// TIA Portal project "Semaforo V2" (V17)

(* hardware
DEVICE "S7-400 station_1"  S7-400 station
   slot 0: "UR1_0"  UR1  6ES7 400-1TA01-0AA0
   slot 1: "PS 407 4A_1"  PS 407 4A  6ES7 407-0DA02-0AA0
   slot 2: "PLC_1"  CPU 416-3 PN/DP  6ES7 416-3ES07-0AB0  V7.0
      slot 2: "MPI/DP interface_1"  X1
      slot 5: "PROFINET interface_1"  PN-IO
         slot 1: "Port_1"  Port
         slot 2: "Port_2"  Port
*)

// ===== PLC "PLC_1"  CPU 416-3 PN/DP =====

VAR_GLOBAL   // PLC tag table "Default tag table"
   "Tag_1" AT %I0.0 : Bool;
   "Tag_2" AT %Q0.0 : Bool;
   "Tag_3" AT %Q0.1 : Bool;
   "Tag_4" AT %Q0.2 : Bool;
   "Tag_5" AT %Q0.6 : Bool;
   "Tag_6" AT %Q0.5 : Bool;
   "Tag_7" AT %Q0.4 : Bool;
   "Tag_8" AT %Q0.3 : Bool;
   "Tag_9" AT %Q0.7 : Bool;
   "Tag_10" AT %M0.0 : Bool;
   "Tag_11" AT %M0.1 : Bool;
   "Tag_12" AT %I0.1 : Bool;
   "Tag_13" AT %M0.2 : Bool;
   "Tag_14" AT %M0.4 : Bool;
   "Pisca" AT %M1.5 : Bool;
END_VAR

DATA_BLOCK "Block_STL_DB"   // DB1
{ S7_Optimized_Access := 'FALSE' }
VERSION : 0.1
// stored: InstanceOfName Block_STL
"Block_STL"
BEGIN
END_DATA_BLOCK

FUNCTION_BLOCK "Block_STL"   // FB1, STL
{ S7_Optimized_Access := 'FALSE' }
VERSION : 0.1
   VAR_INPUT
      Liga_Desliga : Bool;
      Botao_Pedestre : Bool;
   END_VAR
   VAR_OUTPUT
      A_Vermelho : Bool;
      A_Amarelo : Bool;
      A_Verde : Bool;
      B_Vermelho : Bool;
      B_Amarelo : Bool;
      B_Verde : Bool;
      P_Vermelho : Bool;
      P_Verde : Bool;
   END_VAR
   VAR_TEMP
      Jump : Bool;
      Pedestre1 : Bool;
   END_VAR
BEGIN

REGION Network 1: Semaforos Veículos
         A     #Liga_Desliga;
         AN    "TON5".Q;
         =     "TON2".IN;

         S     #A_Verde;
         S     #B_Vermelho;
         S     #P_Vermelho;

         CALL  TON , "TON2"
         ( IN := ,
           PT := T#20S,
           Q  := ,
           ET :=
         );

         A     "TON2".Q;
         R     #A_Verde;
         S     #A_Amarelo;

         CALL  TON, "TON3"
         ( IN := "TON2".Q,
           PT := T#3S,
           Q  := ,
           ET :=
         );

         A     "TON3".Q;
         R     #A_Amarelo;
         R     #B_Vermelho;
         S     #A_Vermelho;
         S     #B_Verde;

         CALL  TON, "TON4"
         ( IN := "TON3".Q,
           PT := T#20S,
           Q  := ,
           ET :=
         );

         A     "TON4".Q;
         R     #B_Verde;
         S     #B_Amarelo;

         CALL  TON, "TON5"
         ( IN := "TON4".Q,
           PT := T#3S,
           Q  := ,
           ET :=
         );

   //Loop
         AN    #Botao_Pedestre;
         A     "TON5".Q;
         R     #B_Amarelo;
         R     #A_Vermelho;

   //Verificação Pedestre
         A     #Botao_Pedestre;
         A     "TON5".Q;
         =     #Jump;

         A     #Jump;
         JU    pedestre;



   pedestre:S     #Pedestre1;

         A     #Pedestre1;

         S     #A_Vermelho;
         R     #A_Verde;
         R     #A_Amarelo;
         S     #B_Vermelho;
         R     #B_Verde;
         R     #B_Amarelo;
         R     #P_Vermelho;
         S     #P_Verde;


         CALL  TON , "TON6"
         ( IN := #Pedestre1,
           PT := T#20S,
           Q  := ,
           ET :=
         );

         A     "TON6".Q;
         A     "Pisca";
         S     #P_Vermelho;

         A     "TON6".Q;
         AN    "Pisca";
         R     #P_Vermelho;


         A     "TON7".Q;
         S     #P_Vermelho;
         R     #A_Vermelho;
   //   S     #A_Verde
         R     #A_Amarelo;
   //S     #B_Vermelho
         R     #B_Verde;
         R     #B_Amarelo;
         R     #P_Verde;
END_REGION
END_FUNCTION_BLOCK

ORGANIZATION_BLOCK "Main"   // OB1, LAD
TITLE = "Main Program Sweep (Cycle)"
{ S7_Optimized_Access := 'FALSE' }
VERSION : 0.1
   VAR_TEMP
      OB1_EV_CLASS : Byte;   // Bits 0-3 = 1 (Coming event), Bits 4-7 = 1 (Event class 1)
      OB1_SCAN_1 : Byte;   // 1 (Cold restart scan 1 of OB 1), 3 (Scan 2-n of OB 1)
      OB1_PRIORITY : Byte;   // Priority of OB Execution
      OB1_OB_NUMBR : Byte;   // 1 (Organization block 1, OB1)
      OB1_RESERVED_1 : Byte;   // Reserved for system
      OB1_RESERVED_2 : Byte;   // Reserved for system
      OB1_PREV_CYCLE : Int;   // Cycle time of previous OB1 scan (milliseconds)
      OB1_MIN_CYCLE : Int;   // Minimum cycle time of OB1 (milliseconds)
      OB1_MAX_CYCLE : Int;   // Maximum cycle time of OB1 (milliseconds)
      OB1_DATE_TIME : Date_And_Time;   // Date and time OB1 started
   END_VAR
BEGIN

REGION Network 1
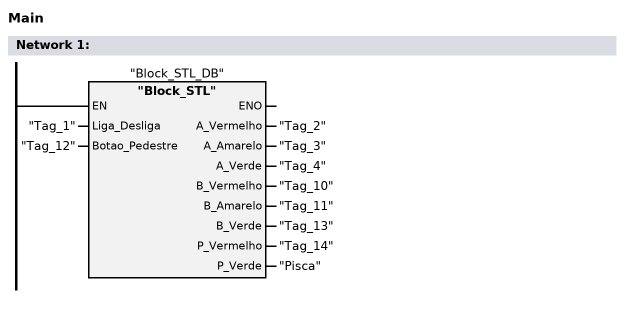
   RUNG wire#powerrail
      "Block_STL_DB"(Liga_Desliga := "Tag_1", Botao_Pedestre := "Tag_12", A_Vermelho => "Tag_2", A_Amarelo => "Tag_3", A_Verde => "Tag_4", B_Vermelho => "Tag_10", B_Amarelo => "Tag_11", B_Verde => "Tag_13", P_Vermelho => "Tag_14", P_Verde => "Pisca")
   END_RUNG
   // the same network as SCL:
   "Block_STL_DB"(Liga_Desliga := "Tag_1",   // "Block_STL"
                  Botao_Pedestre := "Tag_12",
                  A_Vermelho => "Tag_2",
                  A_Amarelo => "Tag_3",
                  A_Verde => "Tag_4",
                  B_Vermelho => "Tag_10",
                  B_Amarelo => "Tag_11",
                  B_Verde => "Tag_13",
                  P_Vermelho => "Tag_14",
                  P_Verde => "Pisca");
END_REGION
END_ORGANIZATION_BLOCK